// TIA Portal V17 export
// export: Created 2025-06-26T07:49:42.6687813Z, ExportSetting WithDefaults, DisplayName Totally Integrated Automation Portal, DisplayVersion V17 Update 8, DisplayName TIA Portal Openness, DisplayVersion V17 Update 8, DisplayName TIA Portal Version Control Interface, DisplayVersion V17, DisplayName STEP 7 Professional, DisplayVersion V17 Update 8, DisplayName STEP 7 Safety, DisplayVersion V17 Update 6, DisplayName WinCC Advanced, DisplayVersion V17 Update 8
FUNCTION_BLOCK "AlarmManagement"   // FB32, LAD
{ S7_Optimized_Access := 'TRUE' }
VERSION : 0.1
// stored: AutoNumber true, IsIECCheckEnabled false, IsRetainMemResEnabled false, MemoryReserve 0, SetENOAutomatically false, UDAEnableTagReadback false
   VAR
      CriticalAlarm_1000 { ExternalAccessible := 'False'; ExternalVisible := 'False'; ExternalWritable := 'False'} : Bool;   // Contribution from 1000-series
      CriticalAlarm_2000 { ExternalAccessible := 'False'; ExternalVisible := 'False'; ExternalWritable := 'False'} : Bool;   // Contribution from 2000-series
      CriticalAlarm_3000 { ExternalAccessible := 'False'; ExternalVisible := 'False'; ExternalWritable := 'False'} : Bool;   // Contribution from 3000-series
      CriticalAlarm_4000 { ExternalAccessible := 'False'; ExternalVisible := 'False'; ExternalWritable := 'False'} : Bool;   // Contribution from 4000-series
      CriticalAlarm_5000 { ExternalAccessible := 'False'; ExternalVisible := 'False'; ExternalWritable := 'False'} : Bool;   // Contribution from 5000-series
      CriticalAlarm_9000 { ExternalAccessible := 'False'; ExternalVisible := 'False'; ExternalWritable := 'False'} : Bool;   // Contribution from 9000-series
      CommonAlarm_1000 { ExternalAccessible := 'False'; ExternalVisible := 'False'; ExternalWritable := 'False'} : Bool;
      CommonAlarm_2000 { ExternalAccessible := 'False'; ExternalVisible := 'False'; ExternalWritable := 'False'} : Bool;
      CommonAlarm_3000 { ExternalAccessible := 'False'; ExternalVisible := 'False'; ExternalWritable := 'False'} : Bool;
      CommonAlarm_5000 { ExternalAccessible := 'False'; ExternalVisible := 'False'; ExternalWritable := 'False'} : Bool;
      CommonAlarm_9000 { ExternalAccessible := 'False'; ExternalVisible := 'False'; ExternalWritable := 'False'} : Bool;
   END_VAR
BEGIN

REGION Network 1 (SCL): Comments
   (*
   This is done with ladder code instead of bits in an alarm struct, so that:
   a) it is easy to see at a glance which alarms are part of the critical alarm (and when monitoring, which alarms are causing the critical alarm)
   b) alarms cannot be removed from the critical alarm by accidentally flipping a bit in a struct, only via code change

   When adding alarms, please add into the correct group and keep each group ordered by alarm number. You will thank yourself later.
   It is easy to make a mess here, resist the urge!
   *)
END_REGION

REGION Network 2: Critical Alarm 1000
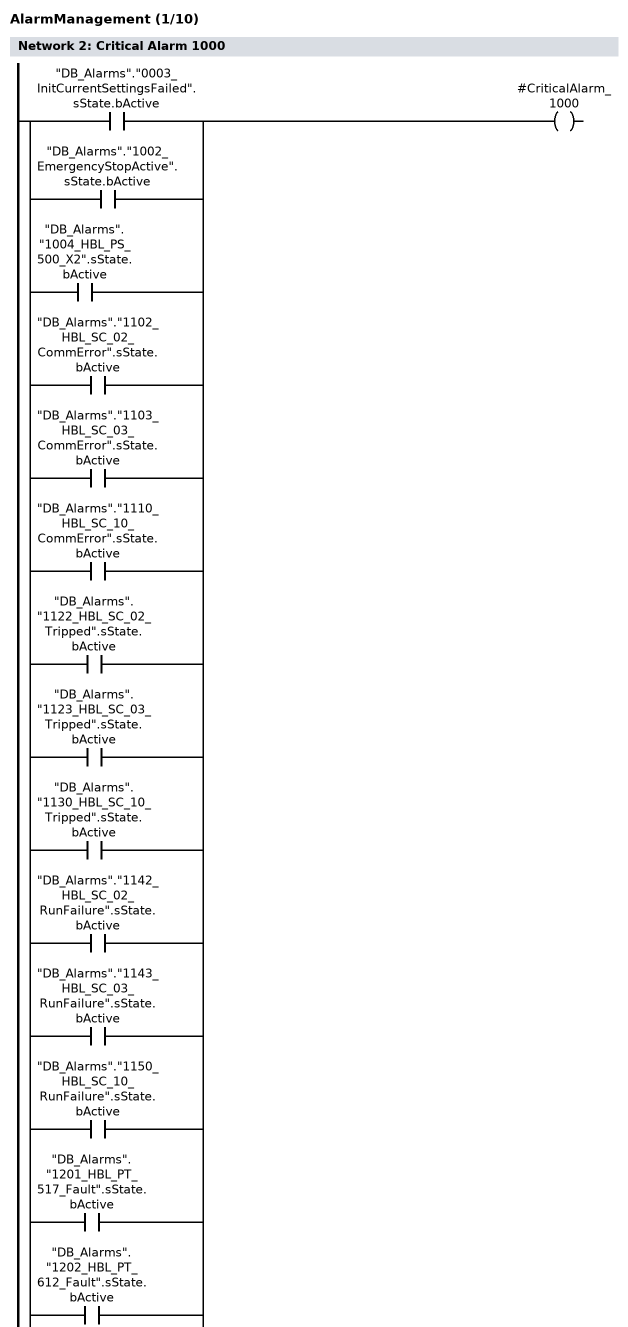
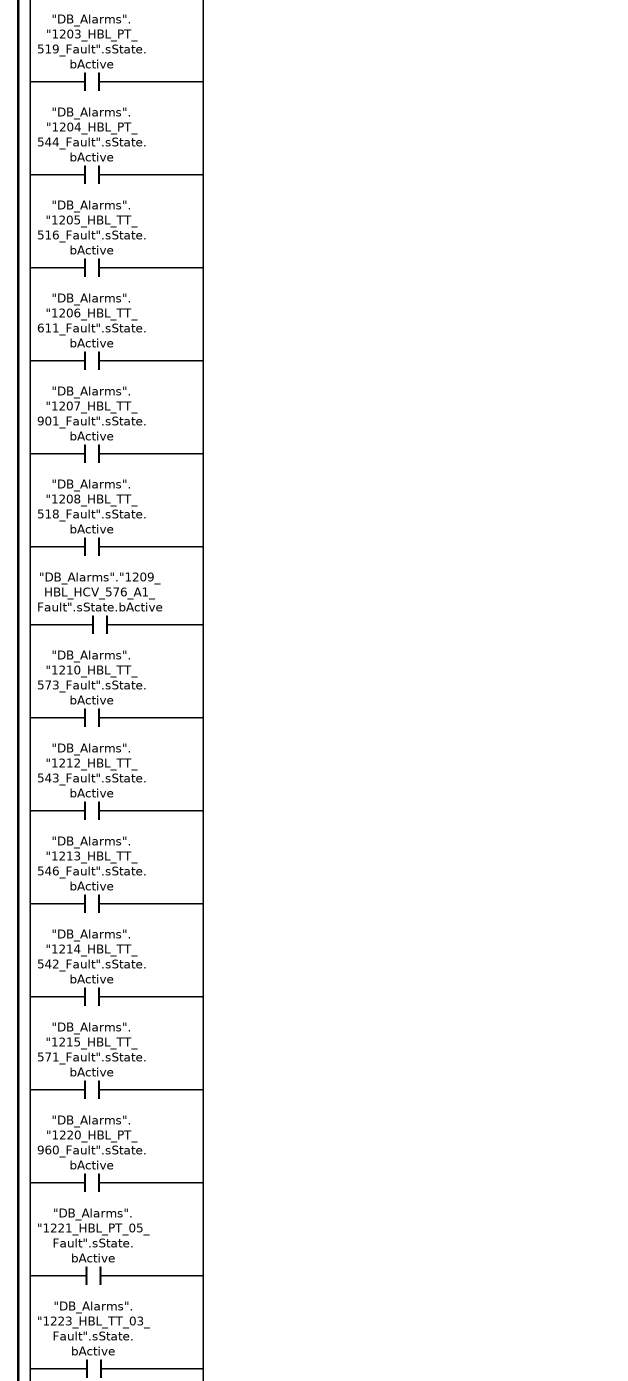
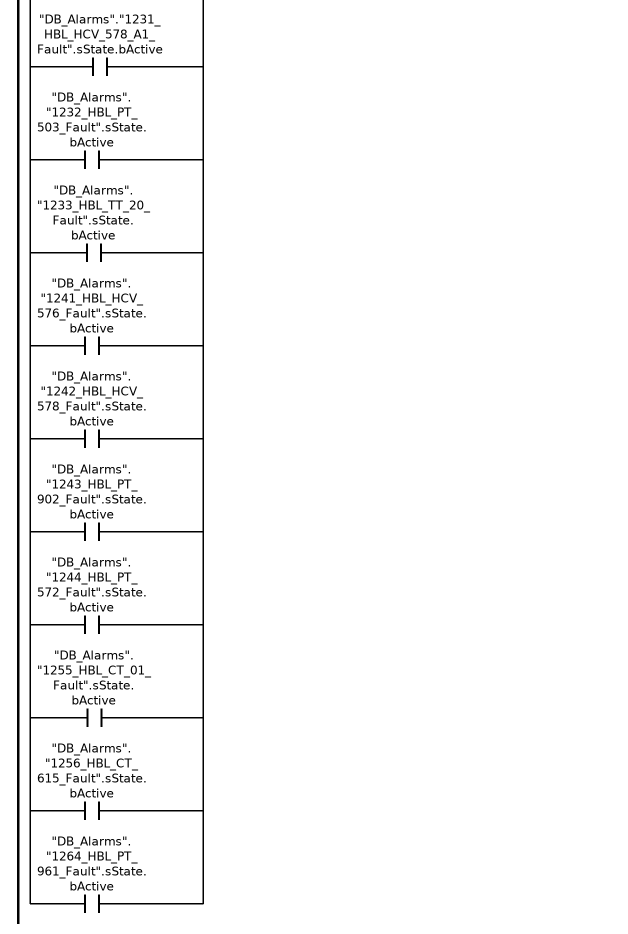
   RUNG wire#powerrail
      Contact( "DB_Alarms"."0003_InitCurrentSettingsFailed".sState.bActive )
      wire#w1
      Coil( #CriticalAlarm_1000 )
   END_RUNG
   RUNG wire#powerrail
      Contact( "DB_Alarms"."1002_EmergencyStopActive".sState.bActive )
   END_RUNG wire#w1
   RUNG wire#powerrail
      Contact( "DB_Alarms"."1004_HBL_PS_500_X2".sState.bActive )
   END_RUNG wire#w1
   RUNG wire#powerrail
      Contact( "DB_Alarms"."1102_HBL_SC_02_CommError".sState.bActive )
   END_RUNG wire#w1
   RUNG wire#powerrail
      Contact( "DB_Alarms"."1103_HBL_SC_03_CommError".sState.bActive )
   END_RUNG wire#w1
   RUNG wire#powerrail
      Contact( "DB_Alarms"."1110_HBL_SC_10_CommError".sState.bActive )
   END_RUNG wire#w1
   RUNG wire#powerrail
      Contact( "DB_Alarms"."1122_HBL_SC_02_Tripped".sState.bActive )
   END_RUNG wire#w1
   RUNG wire#powerrail
      Contact( "DB_Alarms"."1123_HBL_SC_03_Tripped".sState.bActive )
   END_RUNG wire#w1
   RUNG wire#powerrail
      Contact( "DB_Alarms"."1130_HBL_SC_10_Tripped".sState.bActive )
   END_RUNG wire#w1
   RUNG wire#powerrail
      Contact( "DB_Alarms"."1142_HBL_SC_02_RunFailure".sState.bActive )
   END_RUNG wire#w1
   RUNG wire#powerrail
      Contact( "DB_Alarms"."1143_HBL_SC_03_RunFailure".sState.bActive )
   END_RUNG wire#w1
   RUNG wire#powerrail
      Contact( "DB_Alarms"."1150_HBL_SC_10_RunFailure".sState.bActive )
   END_RUNG wire#w1
   RUNG wire#powerrail
      Contact( "DB_Alarms"."1201_HBL_PT_517_Fault".sState.bActive )
   END_RUNG wire#w1
   RUNG wire#powerrail
      Contact( "DB_Alarms"."1202_HBL_PT_612_Fault".sState.bActive )
   END_RUNG wire#w1
   RUNG wire#powerrail
      Contact( "DB_Alarms"."1203_HBL_PT_519_Fault".sState.bActive )
   END_RUNG wire#w1
   RUNG wire#powerrail
      Contact( "DB_Alarms"."1204_HBL_PT_544_Fault".sState.bActive )
   END_RUNG wire#w1
   RUNG wire#powerrail
      Contact( "DB_Alarms"."1205_HBL_TT_516_Fault".sState.bActive )
   END_RUNG wire#w1
   RUNG wire#powerrail
      Contact( "DB_Alarms"."1206_HBL_TT_611_Fault".sState.bActive )
   END_RUNG wire#w1
   RUNG wire#powerrail
      Contact( "DB_Alarms"."1207_HBL_TT_901_Fault".sState.bActive )
   END_RUNG wire#w1
   RUNG wire#powerrail
      Contact( "DB_Alarms"."1208_HBL_TT_518_Fault".sState.bActive )
   END_RUNG wire#w1
   RUNG wire#powerrail
      Contact( "DB_Alarms"."1209_HBL_HCV_576_A1_Fault".sState.bActive )
   END_RUNG wire#w1
   RUNG wire#powerrail
      Contact( "DB_Alarms"."1210_HBL_TT_573_Fault".sState.bActive )
   END_RUNG wire#w1
   RUNG wire#powerrail
      Contact( "DB_Alarms"."1212_HBL_TT_543_Fault".sState.bActive )
   END_RUNG wire#w1
   RUNG wire#powerrail
      Contact( "DB_Alarms"."1213_HBL_TT_546_Fault".sState.bActive )
   END_RUNG wire#w1
   RUNG wire#powerrail
      Contact( "DB_Alarms"."1214_HBL_TT_542_Fault".sState.bActive )
   END_RUNG wire#w1
   RUNG wire#powerrail
      Contact( "DB_Alarms"."1215_HBL_TT_571_Fault".sState.bActive )
   END_RUNG wire#w1
   RUNG wire#powerrail
      Contact( "DB_Alarms"."1220_HBL_PT_960_Fault".sState.bActive )
   END_RUNG wire#w1
   RUNG wire#powerrail
      Contact( "DB_Alarms"."1221_HBL_PT_05_Fault".sState.bActive )
   END_RUNG wire#w1
   RUNG wire#powerrail
      Contact( "DB_Alarms"."1223_HBL_TT_03_Fault".sState.bActive )
   END_RUNG wire#w1
   RUNG wire#powerrail
      Contact( "DB_Alarms"."1231_HBL_HCV_578_A1_Fault".sState.bActive )
   END_RUNG wire#w1
   RUNG wire#powerrail
      Contact( "DB_Alarms"."1232_HBL_PT_503_Fault".sState.bActive )
   END_RUNG wire#w1
   RUNG wire#powerrail
      Contact( "DB_Alarms"."1233_HBL_TT_20_Fault".sState.bActive )
   END_RUNG wire#w1
   RUNG wire#powerrail
      Contact( "DB_Alarms"."1241_HBL_HCV_576_Fault".sState.bActive )
   END_RUNG wire#w1
   RUNG wire#powerrail
      Contact( "DB_Alarms"."1242_HBL_HCV_578_Fault".sState.bActive )
   END_RUNG wire#w1
   RUNG wire#powerrail
      Contact( "DB_Alarms"."1243_HBL_PT_902_Fault".sState.bActive )
   END_RUNG wire#w1
   RUNG wire#powerrail
      Contact( "DB_Alarms"."1244_HBL_PT_572_Fault".sState.bActive )
   END_RUNG wire#w1
   RUNG wire#powerrail
      Contact( "DB_Alarms"."1255_HBL_CT_01_Fault".sState.bActive )
   END_RUNG wire#w1
   RUNG wire#powerrail
      Contact( "DB_Alarms"."1256_HBL_CT_615_Fault".sState.bActive )
   END_RUNG wire#w1
   RUNG wire#powerrail
      Contact( "DB_Alarms"."1264_HBL_PT_961_Fault".sState.bActive )
   END_RUNG wire#w1
   // the same network as SCL:
   #CriticalAlarm_1000 := "DB_Alarms"."0003_InitCurrentSettingsFailed".sState.bActive OR "DB_Alarms"."1002_EmergencyStopActive".sState.bActive OR "DB_Alarms"."1004_HBL_PS_500_X2".sState.bActive OR "DB_Alarms"."1102_HBL_SC_02_CommError".sState.bActive OR "DB_Alarms"."1103_HBL_SC_03_CommError".sState.bActive OR "DB_Alarms"."1110_HBL_SC_10_CommError".sState.bActive OR "DB_Alarms"."1122_HBL_SC_02_Tripped".sState.bActive OR "DB_Alarms"."1123_HBL_SC_03_Tripped".sState.bActive OR "DB_Alarms"."1130_HBL_SC_10_Tripped".sState.bActive OR "DB_Alarms"."1142_HBL_SC_02_RunFailure".sState.bActive OR "DB_Alarms"."1143_HBL_SC_03_RunFailure".sState.bActive OR "DB_Alarms"."1150_HBL_SC_10_RunFailure".sState.bActive OR "DB_Alarms"."1201_HBL_PT_517_Fault".sState.bActive OR "DB_Alarms"."1202_HBL_PT_612_Fault".sState.bActive OR "DB_Alarms"."1203_HBL_PT_519_Fault".sState.bActive OR "DB_Alarms"."1204_HBL_PT_544_Fault".sState.bActive OR "DB_Alarms"."1205_HBL_TT_516_Fault".sState.bActive OR "DB_Alarms"."1206_HBL_TT_611_Fault".sState.bActive OR "DB_Alarms"."1207_HBL_TT_901_Fault".sState.bActive OR "DB_Alarms"."1208_HBL_TT_518_Fault".sState.bActive OR "DB_Alarms"."1209_HBL_HCV_576_A1_Fault".sState.bActive OR "DB_Alarms"."1210_HBL_TT_573_Fault".sState.bActive OR "DB_Alarms"."1212_HBL_TT_543_Fault".sState.bActive OR "DB_Alarms"."1213_HBL_TT_546_Fault".sState.bActive OR "DB_Alarms"."1214_HBL_TT_542_Fault".sState.bActive OR "DB_Alarms"."1215_HBL_TT_571_Fault".sState.bActive OR "DB_Alarms"."1220_HBL_PT_960_Fault".sState.bActive OR "DB_Alarms"."1221_HBL_PT_05_Fault".sState.bActive OR "DB_Alarms"."1223_HBL_TT_03_Fault".sState.bActive OR "DB_Alarms"."1231_HBL_HCV_578_A1_Fault".sState.bActive OR "DB_Alarms"."1232_HBL_PT_503_Fault".sState.bActive OR "DB_Alarms"."1233_HBL_TT_20_Fault".sState.bActive OR "DB_Alarms"."1241_HBL_HCV_576_Fault".sState.bActive OR "DB_Alarms"."1242_HBL_HCV_578_Fault".sState.bActive OR "DB_Alarms"."1243_HBL_PT_902_Fault".sState.bActive OR "DB_Alarms"."1244_HBL_PT_572_Fault".sState.bActive OR "DB_Alarms"."1255_HBL_CT_01_Fault".sState.bActive OR "DB_Alarms"."1256_HBL_CT_615_Fault".sState.bActive OR "DB_Alarms"."1264_HBL_PT_961_Fault".sState.bActive;
END_REGION

REGION Network 3: Critical Alarm 2000
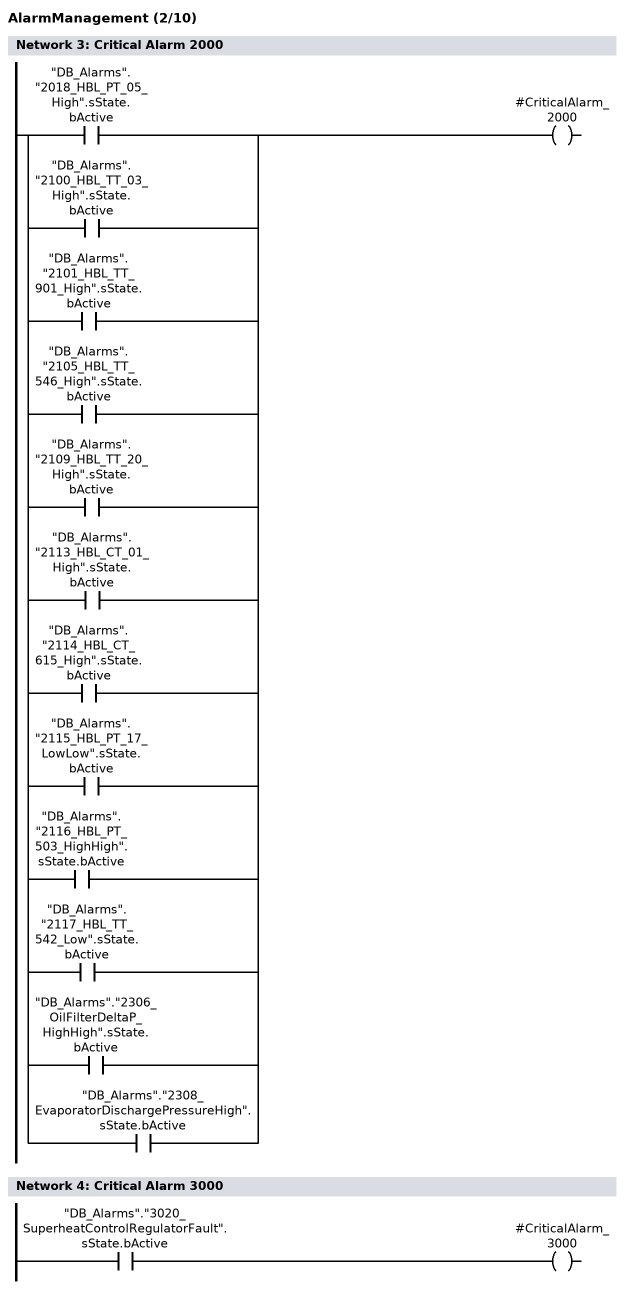
   RUNG wire#powerrail
      Contact( "DB_Alarms"."2018_HBL_PT_05_High".sState.bActive )
      wire#w1
      Coil( #CriticalAlarm_2000 )
   END_RUNG
   RUNG wire#powerrail
      Contact( "DB_Alarms"."2100_HBL_TT_03_High".sState.bActive )
   END_RUNG wire#w1
   RUNG wire#powerrail
      Contact( "DB_Alarms"."2101_HBL_TT_901_High".sState.bActive )
   END_RUNG wire#w1
   RUNG wire#powerrail
      Contact( "DB_Alarms"."2105_HBL_TT_546_High".sState.bActive )
   END_RUNG wire#w1
   RUNG wire#powerrail
      Contact( "DB_Alarms"."2109_HBL_TT_20_High".sState.bActive )
   END_RUNG wire#w1
   RUNG wire#powerrail
      Contact( "DB_Alarms"."2113_HBL_CT_01_High".sState.bActive )
   END_RUNG wire#w1
   RUNG wire#powerrail
      Contact( "DB_Alarms"."2114_HBL_CT_615_High".sState.bActive )
   END_RUNG wire#w1
   RUNG wire#powerrail
      Contact( "DB_Alarms"."2115_HBL_PT_17_LowLow".sState.bActive )
   END_RUNG wire#w1
   RUNG wire#powerrail
      Contact( "DB_Alarms"."2116_HBL_PT_503_HighHigh".sState.bActive )
   END_RUNG wire#w1
   RUNG wire#powerrail
      Contact( "DB_Alarms"."2117_HBL_TT_542_Low".sState.bActive )
   END_RUNG wire#w1
   RUNG wire#powerrail
      Contact( "DB_Alarms"."2306_OilFilterDeltaP_HighHigh".sState.bActive )
   END_RUNG wire#w1
   RUNG wire#powerrail
      Contact( "DB_Alarms"."2308_EvaporatorDischargePressureHigh".sState.bActive )
   END_RUNG wire#w1
   // the same network as SCL:
   #CriticalAlarm_2000 := "DB_Alarms"."2018_HBL_PT_05_High".sState.bActive OR "DB_Alarms"."2100_HBL_TT_03_High".sState.bActive OR "DB_Alarms"."2101_HBL_TT_901_High".sState.bActive OR "DB_Alarms"."2105_HBL_TT_546_High".sState.bActive OR "DB_Alarms"."2109_HBL_TT_20_High".sState.bActive OR "DB_Alarms"."2113_HBL_CT_01_High".sState.bActive OR "DB_Alarms"."2114_HBL_CT_615_High".sState.bActive OR "DB_Alarms"."2115_HBL_PT_17_LowLow".sState.bActive OR "DB_Alarms"."2116_HBL_PT_503_HighHigh".sState.bActive OR "DB_Alarms"."2117_HBL_TT_542_Low".sState.bActive OR "DB_Alarms"."2306_OilFilterDeltaP_HighHigh".sState.bActive OR "DB_Alarms"."2308_EvaporatorDischargePressureHigh".sState.bActive;
END_REGION

REGION Network 4: Critical Alarm 3000
   RUNG wire#powerrail
      Contact( "DB_Alarms"."3020_SuperheatControlRegulatorFault".sState.bActive )
      Coil( #CriticalAlarm_3000 )
   END_RUNG
   // the same network as SCL:
   #CriticalAlarm_3000 := "DB_Alarms"."3020_SuperheatControlRegulatorFault".sState.bActive;
END_REGION

REGION Network 5: Critical Alarm 5000
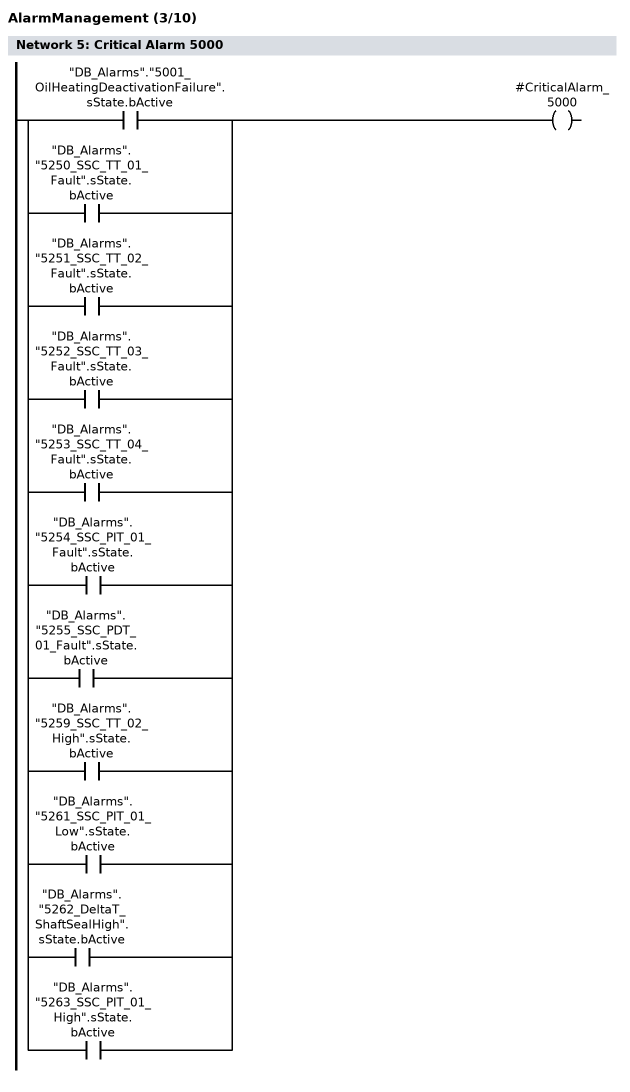
   RUNG wire#powerrail
      Contact( "DB_Alarms"."5001_OilHeatingDeactivationFailure".sState.bActive )
      wire#w1
      Coil( #CriticalAlarm_5000 )
   END_RUNG
   RUNG wire#powerrail
      Contact( "DB_Alarms"."5250_SSC_TT_01_Fault".sState.bActive )
   END_RUNG wire#w1
   RUNG wire#powerrail
      Contact( "DB_Alarms"."5251_SSC_TT_02_Fault".sState.bActive )
   END_RUNG wire#w1
   RUNG wire#powerrail
      Contact( "DB_Alarms"."5252_SSC_TT_03_Fault".sState.bActive )
   END_RUNG wire#w1
   RUNG wire#powerrail
      Contact( "DB_Alarms"."5253_SSC_TT_04_Fault".sState.bActive )
   END_RUNG wire#w1
   RUNG wire#powerrail
      Contact( "DB_Alarms"."5254_SSC_PIT_01_Fault".sState.bActive )
   END_RUNG wire#w1
   RUNG wire#powerrail
      Contact( "DB_Alarms"."5255_SSC_PDT_01_Fault".sState.bActive )
   END_RUNG wire#w1
   RUNG wire#powerrail
      Contact( "DB_Alarms"."5259_SSC_TT_02_High".sState.bActive )
   END_RUNG wire#w1
   RUNG wire#powerrail
      Contact( "DB_Alarms"."5261_SSC_PIT_01_Low".sState.bActive )
   END_RUNG wire#w1
   RUNG wire#powerrail
      Contact( "DB_Alarms"."5262_DeltaT_ShaftSealHigh".sState.bActive )
   END_RUNG wire#w1
   RUNG wire#powerrail
      Contact( "DB_Alarms"."5263_SSC_PIT_01_High".sState.bActive )
   END_RUNG wire#w1
   // the same network as SCL:
   #CriticalAlarm_5000 := "DB_Alarms"."5001_OilHeatingDeactivationFailure".sState.bActive OR "DB_Alarms"."5250_SSC_TT_01_Fault".sState.bActive OR "DB_Alarms"."5251_SSC_TT_02_Fault".sState.bActive OR "DB_Alarms"."5252_SSC_TT_03_Fault".sState.bActive OR "DB_Alarms"."5253_SSC_TT_04_Fault".sState.bActive OR "DB_Alarms"."5254_SSC_PIT_01_Fault".sState.bActive OR "DB_Alarms"."5255_SSC_PDT_01_Fault".sState.bActive OR "DB_Alarms"."5259_SSC_TT_02_High".sState.bActive OR "DB_Alarms"."5261_SSC_PIT_01_Low".sState.bActive OR "DB_Alarms"."5262_DeltaT_ShaftSealHigh".sState.bActive OR "DB_Alarms"."5263_SSC_PIT_01_High".sState.bActive;
END_REGION

REGION Network 6: Critical Alarm 9000
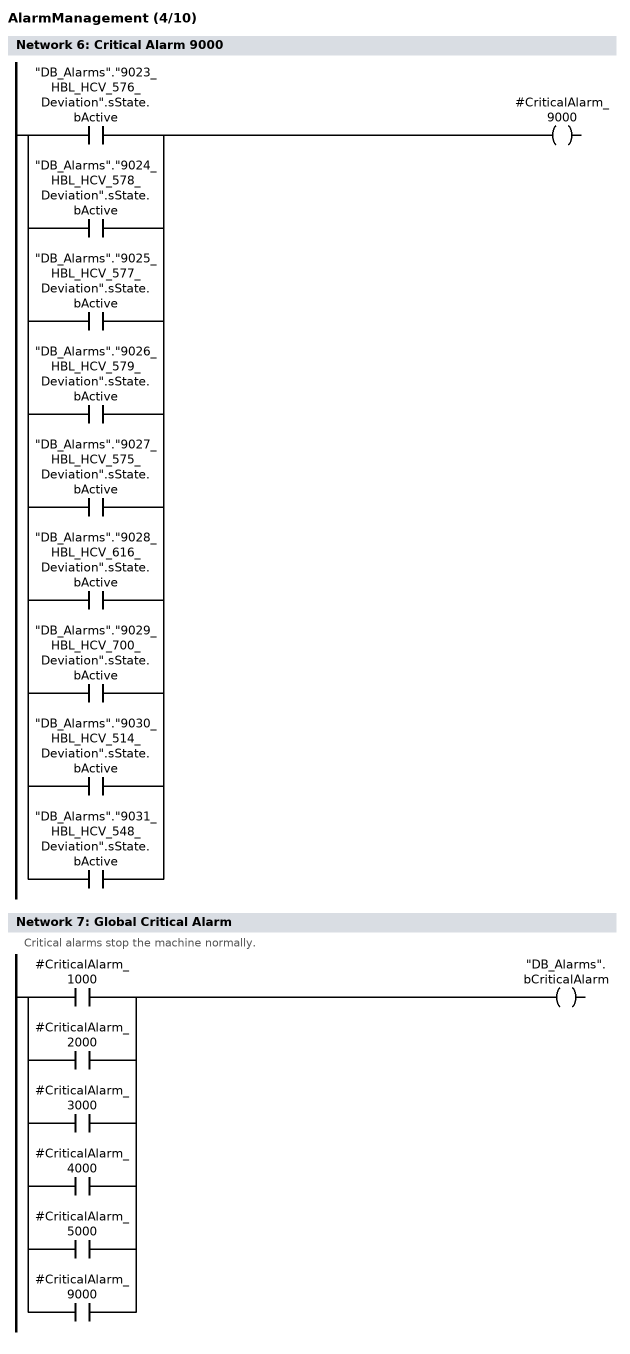
   RUNG wire#powerrail
      Contact( "DB_Alarms"."9023_HBL_HCV_576_Deviation".sState.bActive )
      wire#w1
      Coil( #CriticalAlarm_9000 )
   END_RUNG
   RUNG wire#powerrail
      Contact( "DB_Alarms"."9024_HBL_HCV_578_Deviation".sState.bActive )
   END_RUNG wire#w1
   RUNG wire#powerrail
      Contact( "DB_Alarms"."9025_HBL_HCV_577_Deviation".sState.bActive )
   END_RUNG wire#w1
   RUNG wire#powerrail
      Contact( "DB_Alarms"."9026_HBL_HCV_579_Deviation".sState.bActive )
   END_RUNG wire#w1
   RUNG wire#powerrail
      Contact( "DB_Alarms"."9027_HBL_HCV_575_Deviation".sState.bActive )
   END_RUNG wire#w1
   RUNG wire#powerrail
      Contact( "DB_Alarms"."9028_HBL_HCV_616_Deviation".sState.bActive )
   END_RUNG wire#w1
   RUNG wire#powerrail
      Contact( "DB_Alarms"."9029_HBL_HCV_700_Deviation".sState.bActive )
   END_RUNG wire#w1
   RUNG wire#powerrail
      Contact( "DB_Alarms"."9030_HBL_HCV_514_Deviation".sState.bActive )
   END_RUNG wire#w1
   RUNG wire#powerrail
      Contact( "DB_Alarms"."9031_HBL_HCV_548_Deviation".sState.bActive )
   END_RUNG wire#w1
   // the same network as SCL:
   #CriticalAlarm_9000 := "DB_Alarms"."9023_HBL_HCV_576_Deviation".sState.bActive OR "DB_Alarms"."9024_HBL_HCV_578_Deviation".sState.bActive OR "DB_Alarms"."9025_HBL_HCV_577_Deviation".sState.bActive OR "DB_Alarms"."9026_HBL_HCV_579_Deviation".sState.bActive OR "DB_Alarms"."9027_HBL_HCV_575_Deviation".sState.bActive OR "DB_Alarms"."9028_HBL_HCV_616_Deviation".sState.bActive OR "DB_Alarms"."9029_HBL_HCV_700_Deviation".sState.bActive OR "DB_Alarms"."9030_HBL_HCV_514_Deviation".sState.bActive OR "DB_Alarms"."9031_HBL_HCV_548_Deviation".sState.bActive;
END_REGION

REGION Network 7: Global Critical Alarm
   // Critical alarms stop the machine normally.
   RUNG wire#powerrail
      Contact( #CriticalAlarm_1000 )
      wire#w1
      Coil( "DB_Alarms".bCriticalAlarm )
   END_RUNG
   RUNG wire#powerrail
      Contact( #CriticalAlarm_2000 )
   END_RUNG wire#w1
   RUNG wire#powerrail
      Contact( #CriticalAlarm_3000 )
   END_RUNG wire#w1
   RUNG wire#powerrail
      Contact( #CriticalAlarm_4000 )
   END_RUNG wire#w1
   RUNG wire#powerrail
      Contact( #CriticalAlarm_5000 )
   END_RUNG wire#w1
   RUNG wire#powerrail
      Contact( #CriticalAlarm_9000 )
   END_RUNG wire#w1
   // the same network as SCL:
   "DB_Alarms".bCriticalAlarm := #CriticalAlarm_1000 OR #CriticalAlarm_2000 OR #CriticalAlarm_3000 OR #CriticalAlarm_4000 OR #CriticalAlarm_5000 OR #CriticalAlarm_9000;
END_REGION

REGION Network 8: Common Alarm 1000
   // All alarms that are not critical. Do not activate on critical alarm
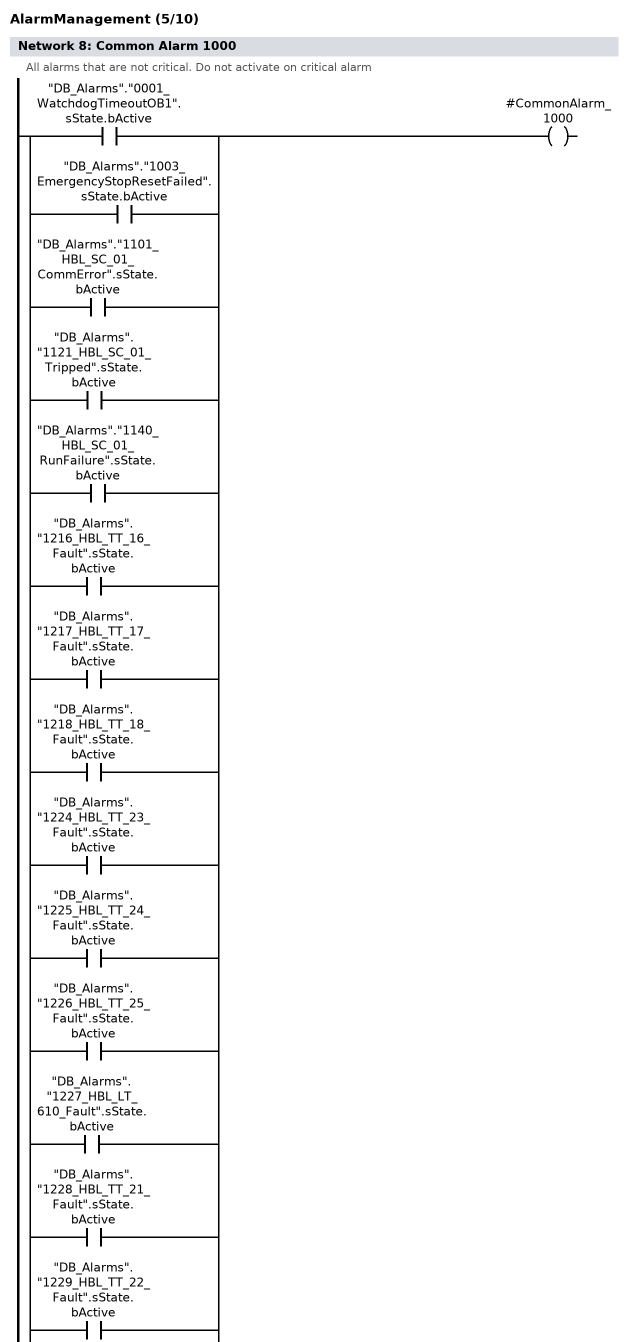
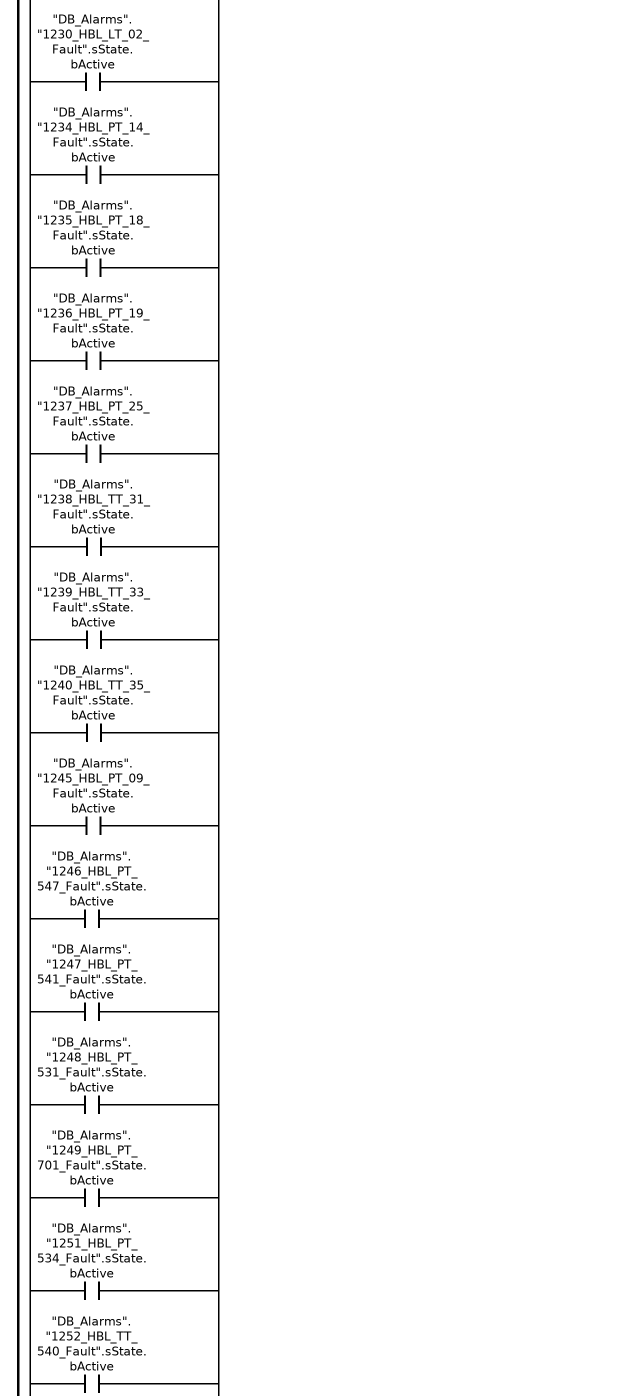
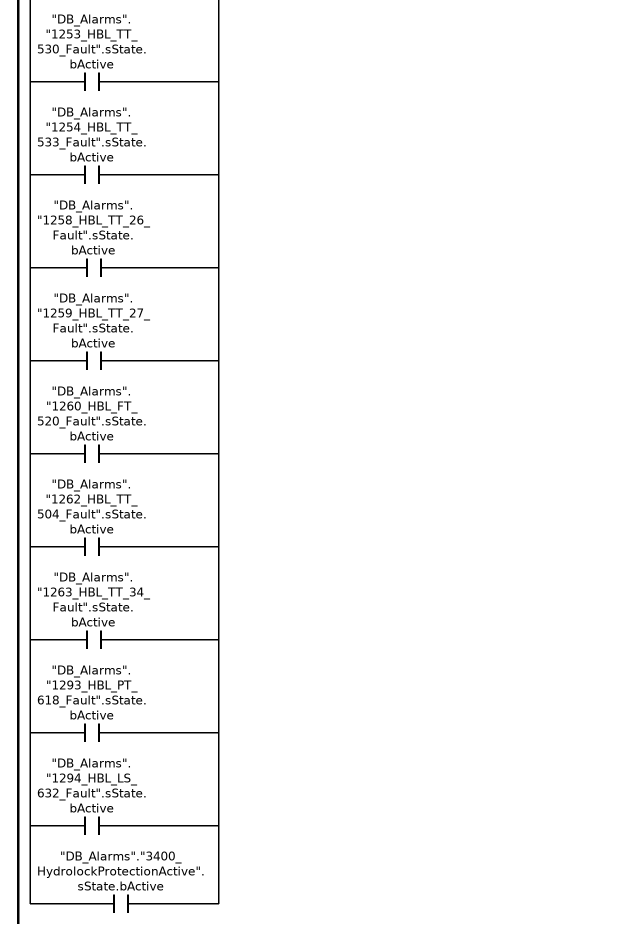
   RUNG wire#powerrail
      Contact( "DB_Alarms"."0001_WatchdogTimeoutOB1".sState.bActive )
      wire#w1
      Coil( #CommonAlarm_1000 )
   END_RUNG
   RUNG wire#powerrail
      Contact( "DB_Alarms"."1003_EmergencyStopResetFailed".sState.bActive )
   END_RUNG wire#w1
   RUNG wire#powerrail
      Contact( "DB_Alarms"."1101_HBL_SC_01_CommError".sState.bActive )
   END_RUNG wire#w1
   RUNG wire#powerrail
      Contact( "DB_Alarms"."1121_HBL_SC_01_Tripped".sState.bActive )
   END_RUNG wire#w1
   RUNG wire#powerrail
      Contact( "DB_Alarms"."1140_HBL_SC_01_RunFailure".sState.bActive )
   END_RUNG wire#w1
   RUNG wire#powerrail
      Contact( "DB_Alarms"."1216_HBL_TT_16_Fault".sState.bActive )
   END_RUNG wire#w1
   RUNG wire#powerrail
      Contact( "DB_Alarms"."1217_HBL_TT_17_Fault".sState.bActive )
   END_RUNG wire#w1
   RUNG wire#powerrail
      Contact( "DB_Alarms"."1218_HBL_TT_18_Fault".sState.bActive )
   END_RUNG wire#w1
   RUNG wire#powerrail
      Contact( "DB_Alarms"."1224_HBL_TT_23_Fault".sState.bActive )
   END_RUNG wire#w1
   RUNG wire#powerrail
      Contact( "DB_Alarms"."1225_HBL_TT_24_Fault".sState.bActive )
   END_RUNG wire#w1
   RUNG wire#powerrail
      Contact( "DB_Alarms"."1226_HBL_TT_25_Fault".sState.bActive )
   END_RUNG wire#w1
   RUNG wire#powerrail
      Contact( "DB_Alarms"."1227_HBL_LT_610_Fault".sState.bActive )
   END_RUNG wire#w1
   RUNG wire#powerrail
      Contact( "DB_Alarms"."1228_HBL_TT_21_Fault".sState.bActive )
   END_RUNG wire#w1
   RUNG wire#powerrail
      Contact( "DB_Alarms"."1229_HBL_TT_22_Fault".sState.bActive )
   END_RUNG wire#w1
   RUNG wire#powerrail
      Contact( "DB_Alarms"."1230_HBL_LT_02_Fault".sState.bActive )
   END_RUNG wire#w1
   RUNG wire#powerrail
      Contact( "DB_Alarms"."1234_HBL_PT_14_Fault".sState.bActive )
   END_RUNG wire#w1
   RUNG wire#powerrail
      Contact( "DB_Alarms"."1235_HBL_PT_18_Fault".sState.bActive )
   END_RUNG wire#w1
   RUNG wire#powerrail
      Contact( "DB_Alarms"."1236_HBL_PT_19_Fault".sState.bActive )
   END_RUNG wire#w1
   RUNG wire#powerrail
      Contact( "DB_Alarms"."1237_HBL_PT_25_Fault".sState.bActive )
   END_RUNG wire#w1
   RUNG wire#powerrail
      Contact( "DB_Alarms"."1238_HBL_TT_31_Fault".sState.bActive )
   END_RUNG wire#w1
   RUNG wire#powerrail
      Contact( "DB_Alarms"."1239_HBL_TT_33_Fault".sState.bActive )
   END_RUNG wire#w1
   RUNG wire#powerrail
      Contact( "DB_Alarms"."1240_HBL_TT_35_Fault".sState.bActive )
   END_RUNG wire#w1
   RUNG wire#powerrail
      Contact( "DB_Alarms"."1245_HBL_PT_09_Fault".sState.bActive )
   END_RUNG wire#w1
   RUNG wire#powerrail
      Contact( "DB_Alarms"."1246_HBL_PT_547_Fault".sState.bActive )
   END_RUNG wire#w1
   RUNG wire#powerrail
      Contact( "DB_Alarms"."1247_HBL_PT_541_Fault".sState.bActive )
   END_RUNG wire#w1
   RUNG wire#powerrail
      Contact( "DB_Alarms"."1248_HBL_PT_531_Fault".sState.bActive )
   END_RUNG wire#w1
   RUNG wire#powerrail
      Contact( "DB_Alarms"."1249_HBL_PT_701_Fault".sState.bActive )
   END_RUNG wire#w1
   RUNG wire#powerrail
      Contact( "DB_Alarms"."1251_HBL_PT_534_Fault".sState.bActive )
   END_RUNG wire#w1
   RUNG wire#powerrail
      Contact( "DB_Alarms"."1252_HBL_TT_540_Fault".sState.bActive )
   END_RUNG wire#w1
   RUNG wire#powerrail
      Contact( "DB_Alarms"."1253_HBL_TT_530_Fault".sState.bActive )
   END_RUNG wire#w1
   RUNG wire#powerrail
      Contact( "DB_Alarms"."1254_HBL_TT_533_Fault".sState.bActive )
   END_RUNG wire#w1
   RUNG wire#powerrail
      Contact( "DB_Alarms"."1258_HBL_TT_26_Fault".sState.bActive )
   END_RUNG wire#w1
   RUNG wire#powerrail
      Contact( "DB_Alarms"."1259_HBL_TT_27_Fault".sState.bActive )
   END_RUNG wire#w1
   RUNG wire#powerrail
      Contact( "DB_Alarms"."1260_HBL_FT_520_Fault".sState.bActive )
   END_RUNG wire#w1
   RUNG wire#powerrail
      Contact( "DB_Alarms"."1262_HBL_TT_504_Fault".sState.bActive )
   END_RUNG wire#w1
   RUNG wire#powerrail
      Contact( "DB_Alarms"."1263_HBL_TT_34_Fault".sState.bActive )
   END_RUNG wire#w1
   RUNG wire#powerrail
      Contact( "DB_Alarms"."1293_HBL_PT_618_Fault".sState.bActive )
   END_RUNG wire#w1
   RUNG wire#powerrail
      Contact( "DB_Alarms"."1294_HBL_LS_632_Fault".sState.bActive )
   END_RUNG wire#w1
   RUNG wire#powerrail
      Contact( "DB_Alarms"."3400_HydrolockProtectionActive".sState.bActive )
   END_RUNG wire#w1
   // the same network as SCL:
   #CommonAlarm_1000 := "DB_Alarms"."0001_WatchdogTimeoutOB1".sState.bActive OR "DB_Alarms"."1003_EmergencyStopResetFailed".sState.bActive OR "DB_Alarms"."1101_HBL_SC_01_CommError".sState.bActive OR "DB_Alarms"."1121_HBL_SC_01_Tripped".sState.bActive OR "DB_Alarms"."1140_HBL_SC_01_RunFailure".sState.bActive OR "DB_Alarms"."1216_HBL_TT_16_Fault".sState.bActive OR "DB_Alarms"."1217_HBL_TT_17_Fault".sState.bActive OR "DB_Alarms"."1218_HBL_TT_18_Fault".sState.bActive OR "DB_Alarms"."1224_HBL_TT_23_Fault".sState.bActive OR "DB_Alarms"."1225_HBL_TT_24_Fault".sState.bActive OR "DB_Alarms"."1226_HBL_TT_25_Fault".sState.bActive OR "DB_Alarms"."1227_HBL_LT_610_Fault".sState.bActive OR "DB_Alarms"."1228_HBL_TT_21_Fault".sState.bActive OR "DB_Alarms"."1229_HBL_TT_22_Fault".sState.bActive OR "DB_Alarms"."1230_HBL_LT_02_Fault".sState.bActive OR "DB_Alarms"."1234_HBL_PT_14_Fault".sState.bActive OR "DB_Alarms"."1235_HBL_PT_18_Fault".sState.bActive OR "DB_Alarms"."1236_HBL_PT_19_Fault".sState.bActive OR "DB_Alarms"."1237_HBL_PT_25_Fault".sState.bActive OR "DB_Alarms"."1238_HBL_TT_31_Fault".sState.bActive OR "DB_Alarms"."1239_HBL_TT_33_Fault".sState.bActive OR "DB_Alarms"."1240_HBL_TT_35_Fault".sState.bActive OR "DB_Alarms"."1245_HBL_PT_09_Fault".sState.bActive OR "DB_Alarms"."1246_HBL_PT_547_Fault".sState.bActive OR "DB_Alarms"."1247_HBL_PT_541_Fault".sState.bActive OR "DB_Alarms"."1248_HBL_PT_531_Fault".sState.bActive OR "DB_Alarms"."1249_HBL_PT_701_Fault".sState.bActive OR "DB_Alarms"."1251_HBL_PT_534_Fault".sState.bActive OR "DB_Alarms"."1252_HBL_TT_540_Fault".sState.bActive OR "DB_Alarms"."1253_HBL_TT_530_Fault".sState.bActive OR "DB_Alarms"."1254_HBL_TT_533_Fault".sState.bActive OR "DB_Alarms"."1258_HBL_TT_26_Fault".sState.bActive OR "DB_Alarms"."1259_HBL_TT_27_Fault".sState.bActive OR "DB_Alarms"."1260_HBL_FT_520_Fault".sState.bActive OR "DB_Alarms"."1262_HBL_TT_504_Fault".sState.bActive OR "DB_Alarms"."1263_HBL_TT_34_Fault".sState.bActive OR "DB_Alarms"."1293_HBL_PT_618_Fault".sState.bActive OR "DB_Alarms"."1294_HBL_LS_632_Fault".sState.bActive OR "DB_Alarms"."3400_HydrolockProtectionActive".sState.bActive;
END_REGION

REGION Network 9: Common Alarm 2000
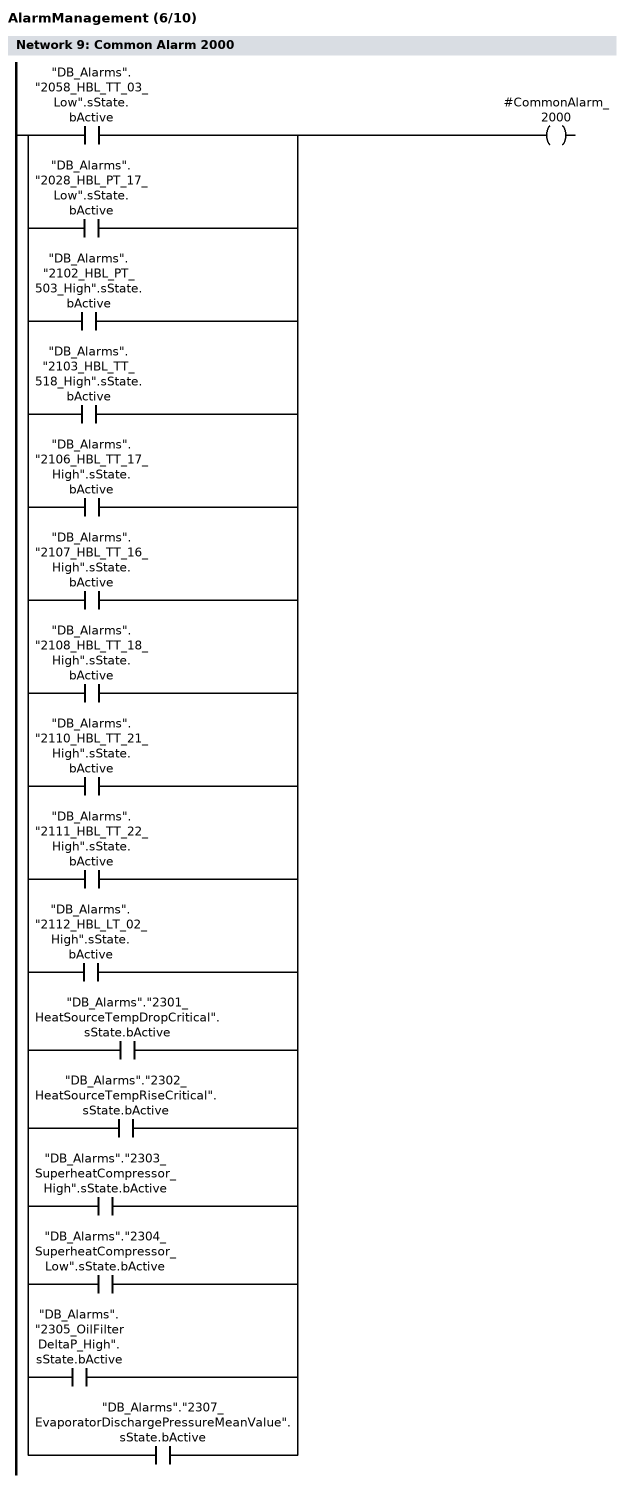
   RUNG wire#powerrail
      Contact( "DB_Alarms"."2058_HBL_TT_03_Low".sState.bActive )
      wire#w1
      Coil( #CommonAlarm_2000 )
   END_RUNG
   RUNG wire#powerrail
      Contact( "DB_Alarms"."2028_HBL_PT_17_Low".sState.bActive )
   END_RUNG wire#w1
   RUNG wire#powerrail
      Contact( "DB_Alarms"."2102_HBL_PT_503_High".sState.bActive )
   END_RUNG wire#w1
   RUNG wire#powerrail
      Contact( "DB_Alarms"."2103_HBL_TT_518_High".sState.bActive )
   END_RUNG wire#w1
   RUNG wire#powerrail
      Contact( "DB_Alarms"."2106_HBL_TT_17_High".sState.bActive )
   END_RUNG wire#w1
   RUNG wire#powerrail
      Contact( "DB_Alarms"."2107_HBL_TT_16_High".sState.bActive )
   END_RUNG wire#w1
   RUNG wire#powerrail
      Contact( "DB_Alarms"."2108_HBL_TT_18_High".sState.bActive )
   END_RUNG wire#w1
   RUNG wire#powerrail
      Contact( "DB_Alarms"."2110_HBL_TT_21_High".sState.bActive )
   END_RUNG wire#w1
   RUNG wire#powerrail
      Contact( "DB_Alarms"."2111_HBL_TT_22_High".sState.bActive )
   END_RUNG wire#w1
   RUNG wire#powerrail
      Contact( "DB_Alarms"."2112_HBL_LT_02_High".sState.bActive )
   END_RUNG wire#w1
   RUNG wire#powerrail
      Contact( "DB_Alarms"."2301_HeatSourceTempDropCritical".sState.bActive )
   END_RUNG wire#w1
   RUNG wire#powerrail
      Contact( "DB_Alarms"."2302_HeatSourceTempRiseCritical".sState.bActive )
   END_RUNG wire#w1
   RUNG wire#powerrail
      Contact( "DB_Alarms"."2303_SuperheatCompressor_High".sState.bActive )
   END_RUNG wire#w1
   RUNG wire#powerrail
      Contact( "DB_Alarms"."2304_SuperheatCompressor_Low".sState.bActive )
   END_RUNG wire#w1
   RUNG wire#powerrail
      Contact( "DB_Alarms"."2305_OilFilterDeltaP_High".sState.bActive )
   END_RUNG wire#w1
   RUNG wire#powerrail
      Contact( "DB_Alarms"."2307_EvaporatorDischargePressureMeanValue".sState.bActive )
   END_RUNG wire#w1
   // the same network as SCL:
   #CommonAlarm_2000 := "DB_Alarms"."2058_HBL_TT_03_Low".sState.bActive OR "DB_Alarms"."2028_HBL_PT_17_Low".sState.bActive OR "DB_Alarms"."2102_HBL_PT_503_High".sState.bActive OR "DB_Alarms"."2103_HBL_TT_518_High".sState.bActive OR "DB_Alarms"."2106_HBL_TT_17_High".sState.bActive OR "DB_Alarms"."2107_HBL_TT_16_High".sState.bActive OR "DB_Alarms"."2108_HBL_TT_18_High".sState.bActive OR "DB_Alarms"."2110_HBL_TT_21_High".sState.bActive OR "DB_Alarms"."2111_HBL_TT_22_High".sState.bActive OR "DB_Alarms"."2112_HBL_LT_02_High".sState.bActive OR "DB_Alarms"."2301_HeatSourceTempDropCritical".sState.bActive OR "DB_Alarms"."2302_HeatSourceTempRiseCritical".sState.bActive OR "DB_Alarms"."2303_SuperheatCompressor_High".sState.bActive OR "DB_Alarms"."2304_SuperheatCompressor_Low".sState.bActive OR "DB_Alarms"."2305_OilFilterDeltaP_High".sState.bActive OR "DB_Alarms"."2307_EvaporatorDischargePressureMeanValue".sState.bActive;
END_REGION

REGION Network 10: Common Alarm 3000
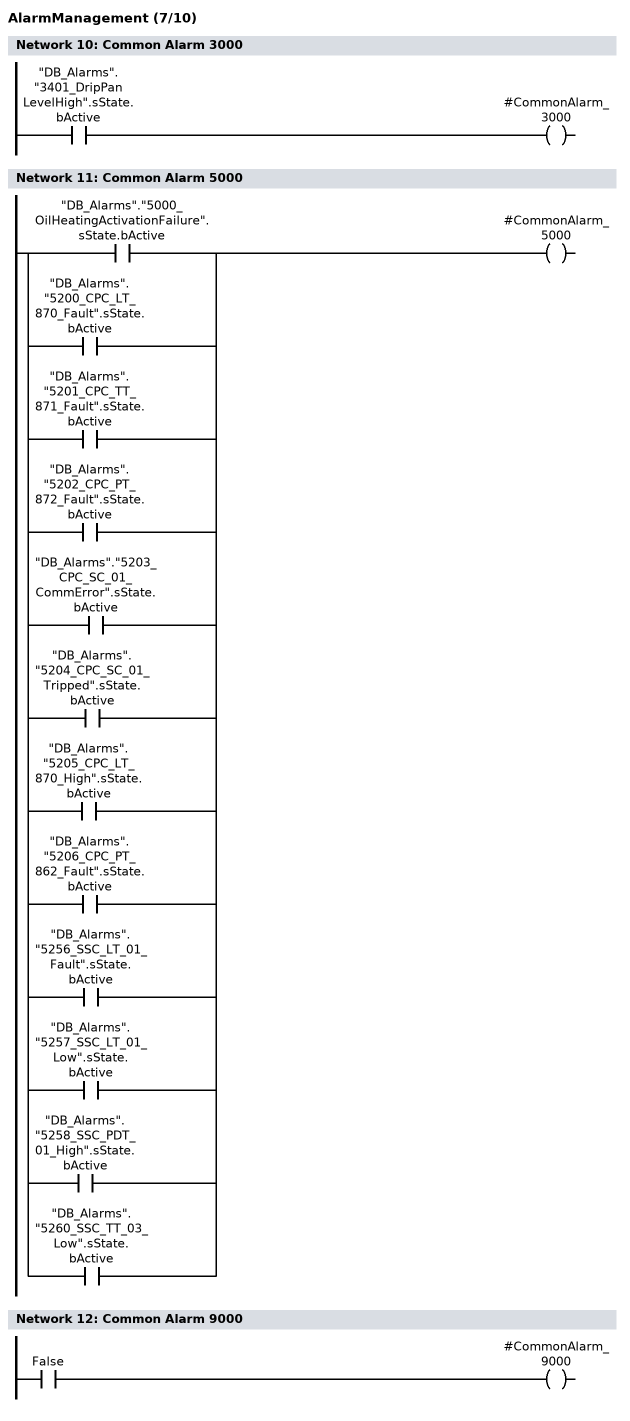
   RUNG wire#powerrail
      Contact( "DB_Alarms"."3401_DripPanLevelHigh".sState.bActive )
      Coil( #CommonAlarm_3000 )
   END_RUNG
   // the same network as SCL:
   #CommonAlarm_3000 := "DB_Alarms"."3401_DripPanLevelHigh".sState.bActive;
END_REGION

REGION Network 11: Common Alarm 5000
   RUNG wire#powerrail
      Contact( "DB_Alarms"."5000_OilHeatingActivationFailure".sState.bActive )
      wire#w1
      Coil( #CommonAlarm_5000 )
   END_RUNG
   RUNG wire#powerrail
      Contact( "DB_Alarms"."5200_CPC_LT_870_Fault".sState.bActive )
   END_RUNG wire#w1
   RUNG wire#powerrail
      Contact( "DB_Alarms"."5201_CPC_TT_871_Fault".sState.bActive )
   END_RUNG wire#w1
   RUNG wire#powerrail
      Contact( "DB_Alarms"."5202_CPC_PT_872_Fault".sState.bActive )
   END_RUNG wire#w1
   RUNG wire#powerrail
      Contact( "DB_Alarms"."5203_CPC_SC_01_CommError".sState.bActive )
   END_RUNG wire#w1
   RUNG wire#powerrail
      Contact( "DB_Alarms"."5204_CPC_SC_01_Tripped".sState.bActive )
   END_RUNG wire#w1
   RUNG wire#powerrail
      Contact( "DB_Alarms"."5205_CPC_LT_870_High".sState.bActive )
   END_RUNG wire#w1
   RUNG wire#powerrail
      Contact( "DB_Alarms"."5206_CPC_PT_862_Fault".sState.bActive )
   END_RUNG wire#w1
   RUNG wire#powerrail
      Contact( "DB_Alarms"."5256_SSC_LT_01_Fault".sState.bActive )
   END_RUNG wire#w1
   RUNG wire#powerrail
      Contact( "DB_Alarms"."5257_SSC_LT_01_Low".sState.bActive )
   END_RUNG wire#w1
   RUNG wire#powerrail
      Contact( "DB_Alarms"."5258_SSC_PDT_01_High".sState.bActive )
   END_RUNG wire#w1
   RUNG wire#powerrail
      Contact( "DB_Alarms"."5260_SSC_TT_03_Low".sState.bActive )
   END_RUNG wire#w1
   // the same network as SCL:
   #CommonAlarm_5000 := "DB_Alarms"."5000_OilHeatingActivationFailure".sState.bActive OR "DB_Alarms"."5200_CPC_LT_870_Fault".sState.bActive OR "DB_Alarms"."5201_CPC_TT_871_Fault".sState.bActive OR "DB_Alarms"."5202_CPC_PT_872_Fault".sState.bActive OR "DB_Alarms"."5203_CPC_SC_01_CommError".sState.bActive OR "DB_Alarms"."5204_CPC_SC_01_Tripped".sState.bActive OR "DB_Alarms"."5205_CPC_LT_870_High".sState.bActive OR "DB_Alarms"."5206_CPC_PT_862_Fault".sState.bActive OR "DB_Alarms"."5256_SSC_LT_01_Fault".sState.bActive OR "DB_Alarms"."5257_SSC_LT_01_Low".sState.bActive OR "DB_Alarms"."5258_SSC_PDT_01_High".sState.bActive OR "DB_Alarms"."5260_SSC_TT_03_Low".sState.bActive;
END_REGION

REGION Network 12: Common Alarm 9000
   RUNG wire#powerrail
      Contact( False )
      Coil( #CommonAlarm_9000 )
   END_RUNG
   // the same network as SCL:
   #CommonAlarm_9000 := False;
END_REGION

REGION Network 13: Global common alarm
   // Alarms do not stop the machine.
   // Alarms in this group are not in the Critical Alarm group
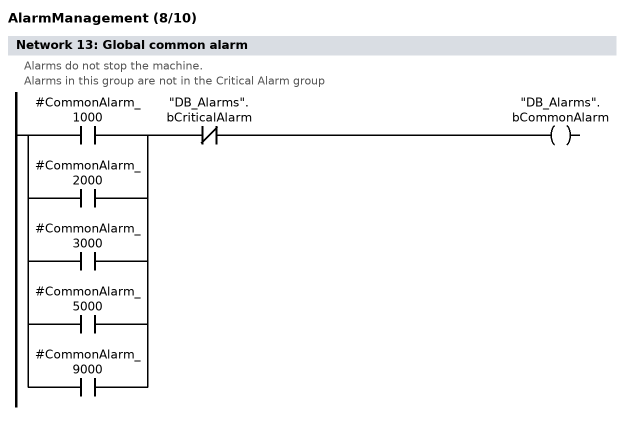
   RUNG wire#powerrail
      Contact( #CommonAlarm_1000 )
      wire#w1
      I_Contact( "DB_Alarms".bCriticalAlarm )
      Coil( "DB_Alarms".bCommonAlarm )
   END_RUNG
   RUNG wire#powerrail
      Contact( #CommonAlarm_2000 )
   END_RUNG wire#w1
   RUNG wire#powerrail
      Contact( #CommonAlarm_3000 )
   END_RUNG wire#w1
   RUNG wire#powerrail
      Contact( #CommonAlarm_5000 )
   END_RUNG wire#w1
   RUNG wire#powerrail
      Contact( #CommonAlarm_9000 )
   END_RUNG wire#w1
   // the same network as SCL:
   "DB_Alarms".bCommonAlarm := (#CommonAlarm_1000 OR #CommonAlarm_2000 OR #CommonAlarm_3000 OR #CommonAlarm_5000 OR #CommonAlarm_9000) AND NOT "DB_Alarms".bCriticalAlarm;
END_REGION

REGION Network 14: FastStop
   // Some critical alarms cause a fast stop, a middle ground between a regular shutdown and an emergency stop
   // All alarms in this group should also be in the Critical Alarms list.
   // The machine shuts down normally but with a faster ramp. See FB34.
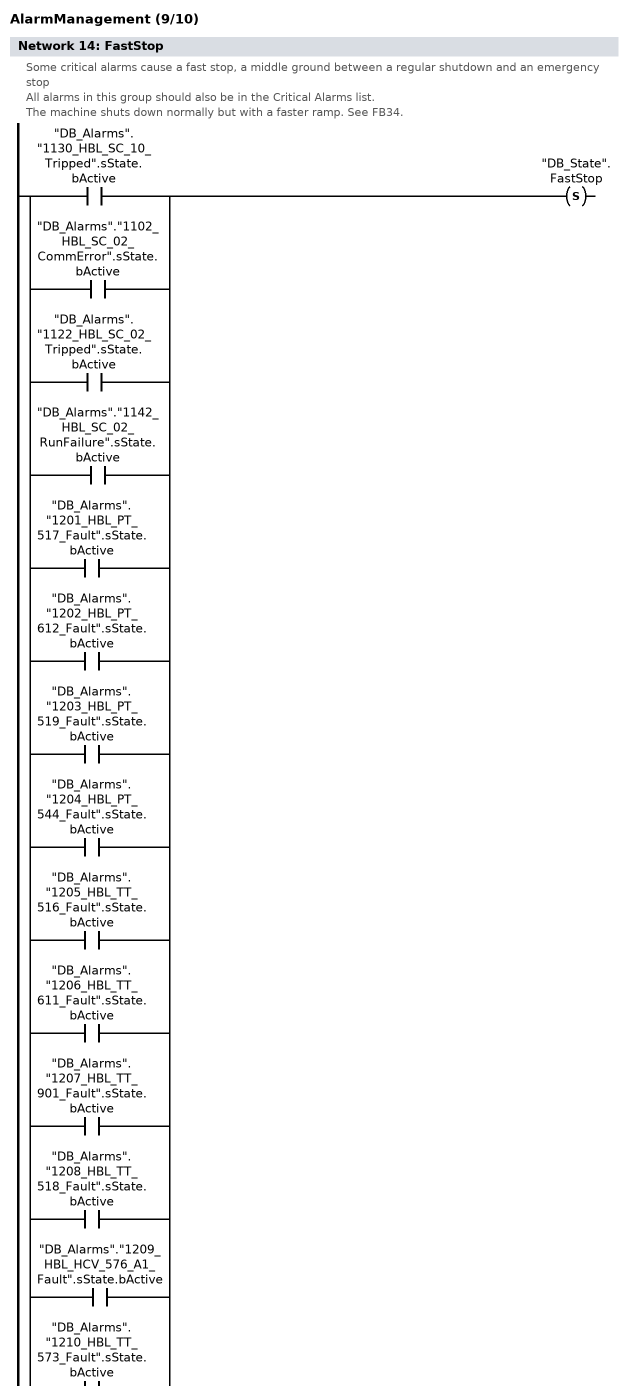
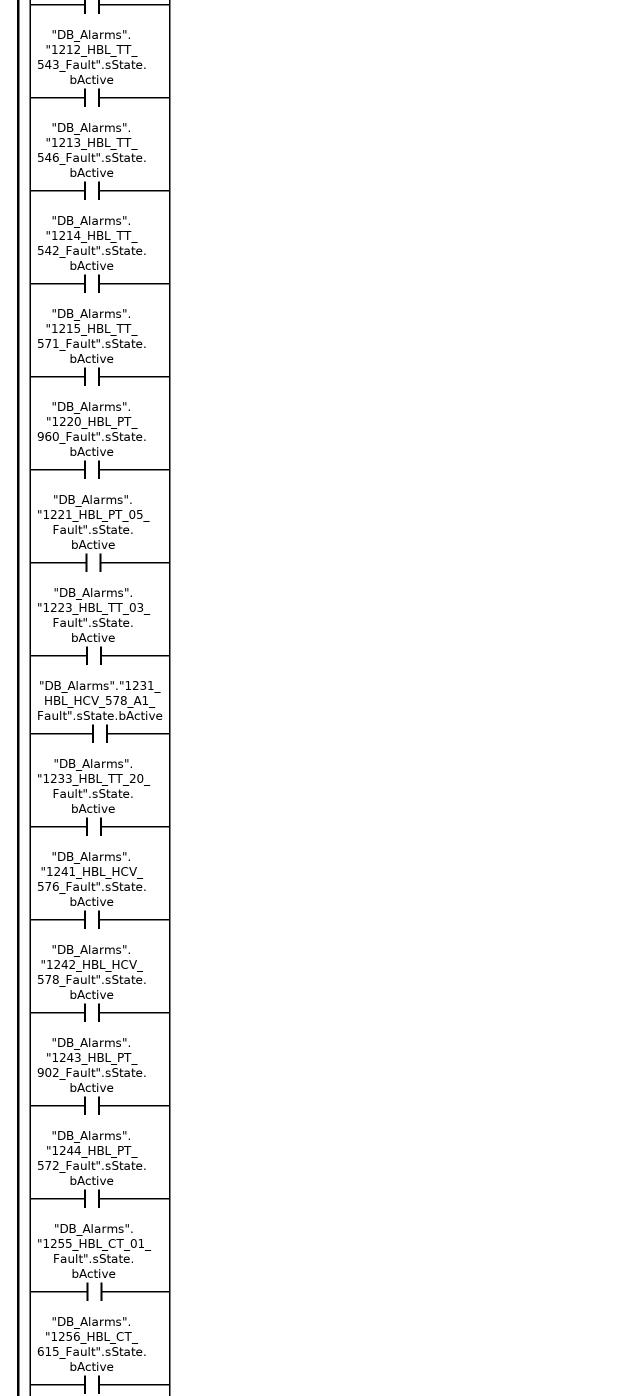
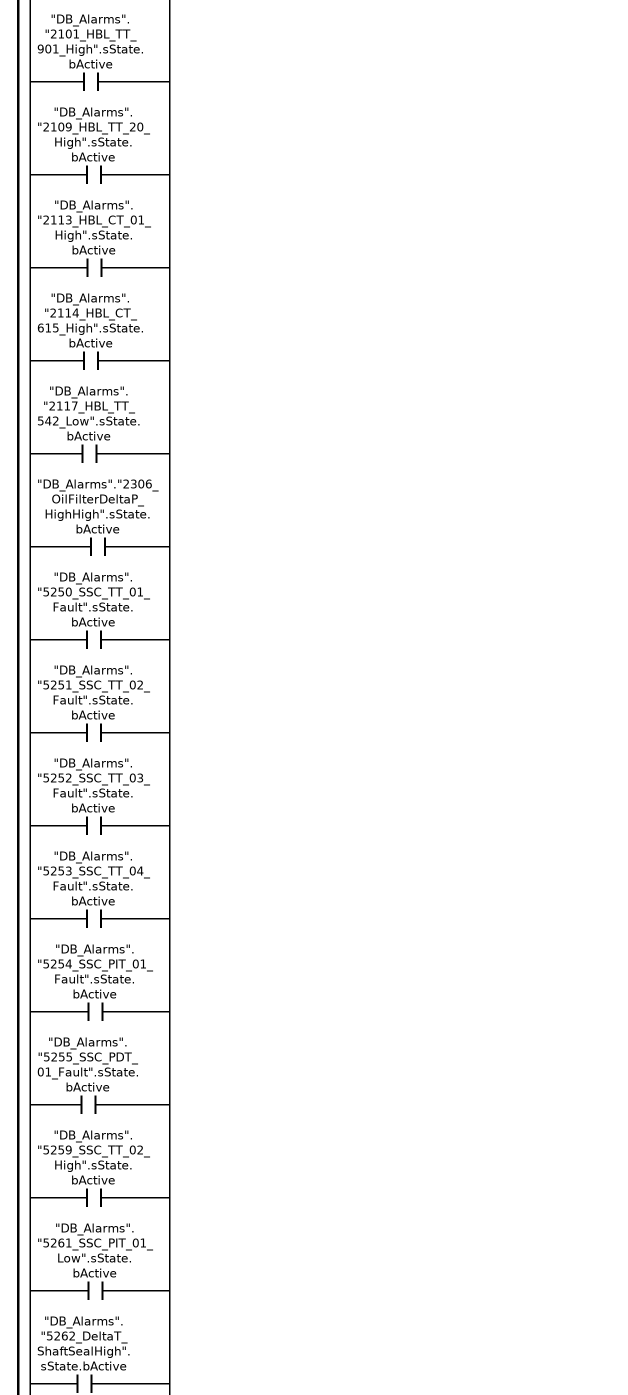
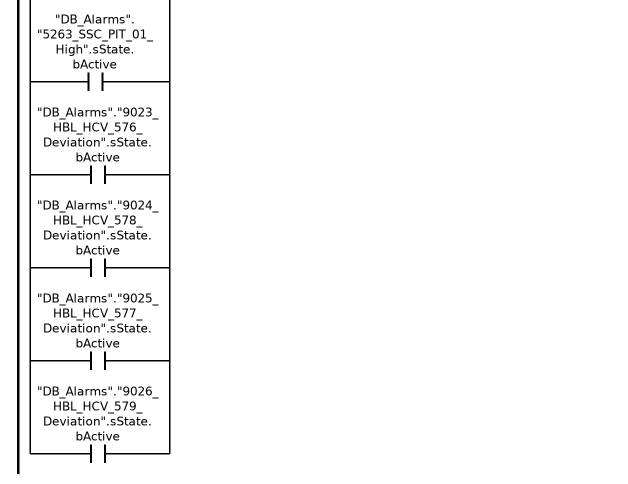
   RUNG wire#powerrail
      Contact( "DB_Alarms"."1130_HBL_SC_10_Tripped".sState.bActive )
      wire#w1
      S_Coil( "DB_State".FastStop )
   END_RUNG
   RUNG wire#powerrail
      Contact( "DB_Alarms"."1102_HBL_SC_02_CommError".sState.bActive )
   END_RUNG wire#w1
   RUNG wire#powerrail
      Contact( "DB_Alarms"."1122_HBL_SC_02_Tripped".sState.bActive )
   END_RUNG wire#w1
   RUNG wire#powerrail
      Contact( "DB_Alarms"."1142_HBL_SC_02_RunFailure".sState.bActive )
   END_RUNG wire#w1
   RUNG wire#powerrail
      Contact( "DB_Alarms"."1201_HBL_PT_517_Fault".sState.bActive )
   END_RUNG wire#w1
   RUNG wire#powerrail
      Contact( "DB_Alarms"."1202_HBL_PT_612_Fault".sState.bActive )
   END_RUNG wire#w1
   RUNG wire#powerrail
      Contact( "DB_Alarms"."1203_HBL_PT_519_Fault".sState.bActive )
   END_RUNG wire#w1
   RUNG wire#powerrail
      Contact( "DB_Alarms"."1204_HBL_PT_544_Fault".sState.bActive )
   END_RUNG wire#w1
   RUNG wire#powerrail
      Contact( "DB_Alarms"."1205_HBL_TT_516_Fault".sState.bActive )
   END_RUNG wire#w1
   RUNG wire#powerrail
      Contact( "DB_Alarms"."1206_HBL_TT_611_Fault".sState.bActive )
   END_RUNG wire#w1
   RUNG wire#powerrail
      Contact( "DB_Alarms"."1207_HBL_TT_901_Fault".sState.bActive )
   END_RUNG wire#w1
   RUNG wire#powerrail
      Contact( "DB_Alarms"."1208_HBL_TT_518_Fault".sState.bActive )
   END_RUNG wire#w1
   RUNG wire#powerrail
      Contact( "DB_Alarms"."1209_HBL_HCV_576_A1_Fault".sState.bActive )
   END_RUNG wire#w1
   RUNG wire#powerrail
      Contact( "DB_Alarms"."1210_HBL_TT_573_Fault".sState.bActive )
   END_RUNG wire#w1
   RUNG wire#powerrail
      Contact( "DB_Alarms"."1212_HBL_TT_543_Fault".sState.bActive )
   END_RUNG wire#w1
   RUNG wire#powerrail
      Contact( "DB_Alarms"."1213_HBL_TT_546_Fault".sState.bActive )
   END_RUNG wire#w1
   RUNG wire#powerrail
      Contact( "DB_Alarms"."1214_HBL_TT_542_Fault".sState.bActive )
   END_RUNG wire#w1
   RUNG wire#powerrail
      Contact( "DB_Alarms"."1215_HBL_TT_571_Fault".sState.bActive )
   END_RUNG wire#w1
   RUNG wire#powerrail
      Contact( "DB_Alarms"."1220_HBL_PT_960_Fault".sState.bActive )
   END_RUNG wire#w1
   RUNG wire#powerrail
      Contact( "DB_Alarms"."1221_HBL_PT_05_Fault".sState.bActive )
   END_RUNG wire#w1
   RUNG wire#powerrail
      Contact( "DB_Alarms"."1223_HBL_TT_03_Fault".sState.bActive )
   END_RUNG wire#w1
   RUNG wire#powerrail
      Contact( "DB_Alarms"."1231_HBL_HCV_578_A1_Fault".sState.bActive )
   END_RUNG wire#w1
   RUNG wire#powerrail
      Contact( "DB_Alarms"."1233_HBL_TT_20_Fault".sState.bActive )
   END_RUNG wire#w1
   RUNG wire#powerrail
      Contact( "DB_Alarms"."1241_HBL_HCV_576_Fault".sState.bActive )
   END_RUNG wire#w1
   RUNG wire#powerrail
      Contact( "DB_Alarms"."1242_HBL_HCV_578_Fault".sState.bActive )
   END_RUNG wire#w1
   RUNG wire#powerrail
      Contact( "DB_Alarms"."1243_HBL_PT_902_Fault".sState.bActive )
   END_RUNG wire#w1
   RUNG wire#powerrail
      Contact( "DB_Alarms"."1244_HBL_PT_572_Fault".sState.bActive )
   END_RUNG wire#w1
   RUNG wire#powerrail
      Contact( "DB_Alarms"."1255_HBL_CT_01_Fault".sState.bActive )
   END_RUNG wire#w1
   RUNG wire#powerrail
      Contact( "DB_Alarms"."1256_HBL_CT_615_Fault".sState.bActive )
   END_RUNG wire#w1
   RUNG wire#powerrail
      Contact( "DB_Alarms"."2101_HBL_TT_901_High".sState.bActive )
   END_RUNG wire#w1
   RUNG wire#powerrail
      Contact( "DB_Alarms"."2109_HBL_TT_20_High".sState.bActive )
   END_RUNG wire#w1
   RUNG wire#powerrail
      Contact( "DB_Alarms"."2113_HBL_CT_01_High".sState.bActive )
   END_RUNG wire#w1
   RUNG wire#powerrail
      Contact( "DB_Alarms"."2114_HBL_CT_615_High".sState.bActive )
   END_RUNG wire#w1
   RUNG wire#powerrail
      Contact( "DB_Alarms"."2117_HBL_TT_542_Low".sState.bActive )
   END_RUNG wire#w1
   RUNG wire#powerrail
      Contact( "DB_Alarms"."2306_OilFilterDeltaP_HighHigh".sState.bActive )
   END_RUNG wire#w1
   RUNG wire#powerrail
      Contact( "DB_Alarms"."5250_SSC_TT_01_Fault".sState.bActive )
   END_RUNG wire#w1
   RUNG wire#powerrail
      Contact( "DB_Alarms"."5251_SSC_TT_02_Fault".sState.bActive )
   END_RUNG wire#w1
   RUNG wire#powerrail
      Contact( "DB_Alarms"."5252_SSC_TT_03_Fault".sState.bActive )
   END_RUNG wire#w1
   RUNG wire#powerrail
      Contact( "DB_Alarms"."5253_SSC_TT_04_Fault".sState.bActive )
   END_RUNG wire#w1
   RUNG wire#powerrail
      Contact( "DB_Alarms"."5254_SSC_PIT_01_Fault".sState.bActive )
   END_RUNG wire#w1
   RUNG wire#powerrail
      Contact( "DB_Alarms"."5255_SSC_PDT_01_Fault".sState.bActive )
   END_RUNG wire#w1
   RUNG wire#powerrail
      Contact( "DB_Alarms"."5259_SSC_TT_02_High".sState.bActive )
   END_RUNG wire#w1
   RUNG wire#powerrail
      Contact( "DB_Alarms"."5261_SSC_PIT_01_Low".sState.bActive )
   END_RUNG wire#w1
   RUNG wire#powerrail
      Contact( "DB_Alarms"."5262_DeltaT_ShaftSealHigh".sState.bActive )
   END_RUNG wire#w1
   RUNG wire#powerrail
      Contact( "DB_Alarms"."5263_SSC_PIT_01_High".sState.bActive )
   END_RUNG wire#w1
   RUNG wire#powerrail
      Contact( "DB_Alarms"."9023_HBL_HCV_576_Deviation".sState.bActive )
   END_RUNG wire#w1
   RUNG wire#powerrail
      Contact( "DB_Alarms"."9024_HBL_HCV_578_Deviation".sState.bActive )
   END_RUNG wire#w1
   RUNG wire#powerrail
      Contact( "DB_Alarms"."9025_HBL_HCV_577_Deviation".sState.bActive )
   END_RUNG wire#w1
   RUNG wire#powerrail
      Contact( "DB_Alarms"."9026_HBL_HCV_579_Deviation".sState.bActive )
   END_RUNG wire#w1
   // the same network as SCL:
   IF "DB_Alarms"."1130_HBL_SC_10_Tripped".sState.bActive OR "DB_Alarms"."1102_HBL_SC_02_CommError".sState.bActive OR "DB_Alarms"."1122_HBL_SC_02_Tripped".sState.bActive OR "DB_Alarms"."1142_HBL_SC_02_RunFailure".sState.bActive OR "DB_Alarms"."1201_HBL_PT_517_Fault".sState.bActive OR "DB_Alarms"."1202_HBL_PT_612_Fault".sState.bActive OR "DB_Alarms"."1203_HBL_PT_519_Fault".sState.bActive OR "DB_Alarms"."1204_HBL_PT_544_Fault".sState.bActive OR "DB_Alarms"."1205_HBL_TT_516_Fault".sState.bActive OR "DB_Alarms"."1206_HBL_TT_611_Fault".sState.bActive OR "DB_Alarms"."1207_HBL_TT_901_Fault".sState.bActive OR "DB_Alarms"."1208_HBL_TT_518_Fault".sState.bActive OR "DB_Alarms"."1209_HBL_HCV_576_A1_Fault".sState.bActive OR "DB_Alarms"."1210_HBL_TT_573_Fault".sState.bActive OR "DB_Alarms"."1212_HBL_TT_543_Fault".sState.bActive OR "DB_Alarms"."1213_HBL_TT_546_Fault".sState.bActive OR "DB_Alarms"."1214_HBL_TT_542_Fault".sState.bActive OR "DB_Alarms"."1215_HBL_TT_571_Fault".sState.bActive OR "DB_Alarms"."1220_HBL_PT_960_Fault".sState.bActive OR "DB_Alarms"."1221_HBL_PT_05_Fault".sState.bActive OR "DB_Alarms"."1223_HBL_TT_03_Fault".sState.bActive OR "DB_Alarms"."1231_HBL_HCV_578_A1_Fault".sState.bActive OR "DB_Alarms"."1233_HBL_TT_20_Fault".sState.bActive OR "DB_Alarms"."1241_HBL_HCV_576_Fault".sState.bActive OR "DB_Alarms"."1242_HBL_HCV_578_Fault".sState.bActive OR "DB_Alarms"."1243_HBL_PT_902_Fault".sState.bActive OR "DB_Alarms"."1244_HBL_PT_572_Fault".sState.bActive OR "DB_Alarms"."1255_HBL_CT_01_Fault".sState.bActive OR "DB_Alarms"."1256_HBL_CT_615_Fault".sState.bActive OR "DB_Alarms"."2101_HBL_TT_901_High".sState.bActive OR "DB_Alarms"."2109_HBL_TT_20_High".sState.bActive OR "DB_Alarms"."2113_HBL_CT_01_High".sState.bActive OR "DB_Alarms"."2114_HBL_CT_615_High".sState.bActive OR "DB_Alarms"."2117_HBL_TT_542_Low".sState.bActive OR "DB_Alarms"."2306_OilFilterDeltaP_HighHigh".sState.bActive OR "DB_Alarms"."5250_SSC_TT_01_Fault".sState.bActive OR "DB_Alarms"."5251_SSC_TT_02_Fault".sState.bActive OR "DB_Alarms"."5252_SSC_TT_03_Fault".sState.bActive OR "DB_Alarms"."5253_SSC_TT_04_Fault".sState.bActive OR "DB_Alarms"."5254_SSC_PIT_01_Fault".sState.bActive OR "DB_Alarms"."5255_SSC_PDT_01_Fault".sState.bActive OR "DB_Alarms"."5259_SSC_TT_02_High".sState.bActive OR "DB_Alarms"."5261_SSC_PIT_01_Low".sState.bActive OR "DB_Alarms"."5262_DeltaT_ShaftSealHigh".sState.bActive OR "DB_Alarms"."5263_SSC_PIT_01_High".sState.bActive OR "DB_Alarms"."9023_HBL_HCV_576_Deviation".sState.bActive OR "DB_Alarms"."9024_HBL_HCV_578_Deviation".sState.bActive OR "DB_Alarms"."9025_HBL_HCV_577_Deviation".sState.bActive OR "DB_Alarms"."9026_HBL_HCV_579_Deviation".sState.bActive THEN
       "DB_State".FastStop := TRUE;
   END_IF;
END_REGION

REGION Network 15: Ack All reset (don't touch)
   // Clear it first
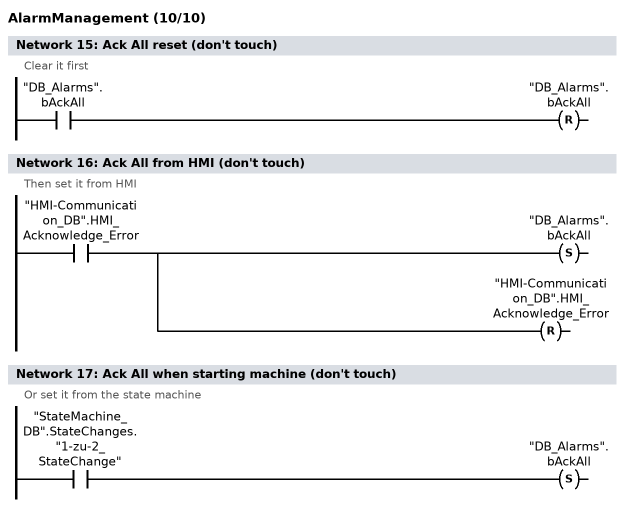
   RUNG wire#powerrail
      Contact( "DB_Alarms".bAckAll )
      R_Coil( "DB_Alarms".bAckAll )
   END_RUNG
   // the same network as SCL:
   IF "DB_Alarms".bAckAll THEN "DB_Alarms".bAckAll := FALSE; END_IF;
END_REGION

REGION Network 16: Ack All from HMI (don't touch)
   // Then set it from HMI
   RUNG wire#powerrail
      Contact( "HMI-Communication_DB".HMI_Acknowledge_Error )
      wire#w1
      S_Coil( "DB_Alarms".bAckAll )
   END_RUNG
   RUNG wire#w1
      R_Coil( "HMI-Communication_DB".HMI_Acknowledge_Error )
   END_RUNG
   // the same network as SCL:
   IF "HMI-Communication_DB".HMI_Acknowledge_Error THEN
       "DB_Alarms".bAckAll := TRUE;
       "HMI-Communication_DB".HMI_Acknowledge_Error := FALSE;
   END_IF;
END_REGION

REGION Network 17: Ack All when starting machine (don't touch)
   // Or set it from the state machine
   RUNG wire#powerrail
      Contact( "StateMachine_DB".StateChanges."1-zu-2_StateChange" )
      S_Coil( "DB_Alarms".bAckAll )
   END_RUNG
   // the same network as SCL:
   IF "StateMachine_DB".StateChanges."1-zu-2_StateChange" THEN "DB_Alarms".bAckAll := TRUE; END_IF;
END_REGION
END_FUNCTION_BLOCK
